TYPE libT_LongSTRING : STRING(1023);
END_TYPE

(* stored: Version 1.1.0.1
   DUT libT_LongSTRING: Id {845ff768-7d91-4814-8251-e2d4c721c106} *)
